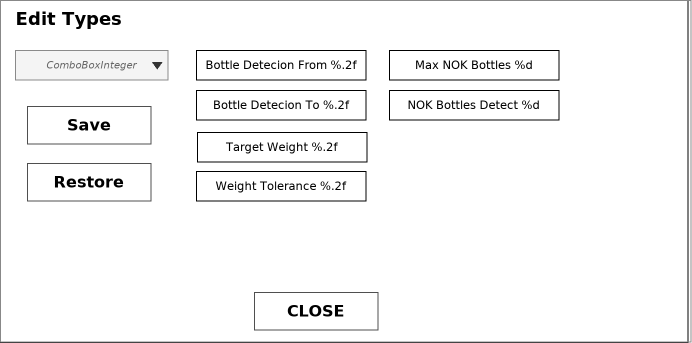
VISUALIZATION vTableEditTypes  // 692x343
VAR_IN_OUT
	fbTableControl: FB_TableControl;
END_VAR
    Rectangle (0,0 688x343)
    Label (-4,2 145x34), "Edit Types"
    Rectangle (254,292 124x38), "CLOSE"
        OnMouseDown: execute { fbTableControl.stHMI.iDialogNumber:=0; }
    ComboBoxInteger (15,50 153x30), variable: fbTableControl.stHMI.nEditedType, text list: 'tlBottleTypes'
    Rectangle (27,106 124x38), "Save"
        OnMouseDown: execute { fbTableControl.stHMI.bSave:=TRUE; }
    Rectangle (196,50 170x30), "Bottle Detecion From %.2f", text variable: fbTableControl.stHMI.stEditedType.stLoadingBottleParams.rLoadingDetectionFrom
        OnMouseClick: write the text variable via Default, min 0, max 32767, title 'Detection From', format %.2f
    Rectangle (196,90 170x30), "Bottle Detecion To %.2f", text variable: fbTableControl.stHMI.stEditedType.stLoadingBottleParams.rLoadingDetectionTo
        OnMouseClick: write the text variable via Default, min 0, max 32767, title 'Detection To', format %.2f
    Rectangle (27,163 124x38), "Restore"
        OnMouseDown: execute { fbTableControl.stHMI.bRestore:=TRUE; }
    Rectangle (197,132 170x30), "Target Weight %.2f", text variable: fbTableControl.stHMI.stEditedType.stWeighingBottleParams.rTargetWeight
        OnMouseClick: write the text variable via Default, min 0, max 2000, title 'Target Weight', format %.2f
    Rectangle (196,171 170x30), "Weight Tolerance %.2f", text variable: fbTableControl.stHMI.stEditedType.stWeighingBottleParams.rWeightTolerance
        OnMouseClick: write the text variable via Default, min 0, max 50, title 'Weight Tolerance', format %.2f
    Rectangle (389,50 170x30), "Max NOK Bottles %d", text variable: fbTableControl.stHMI.stEditedType.stWeighingBottleParams.iMaxNOK_Bottles
        OnMouseClick: write the text variable via Default, min 0, max 50, title 'Weight Tolerance', format %.2f
    Rectangle (389,90 170x30), "NOK Bottles Detect %d", text variable: fbTableControl.stHMI.stEditedType.stWeighingBottleParams.iNOK_BottlesSensorDetect
        OnMouseClick: write the text variable via Default, min 0, max 50, title 'Weight Tolerance', format %.2f
END_VISUALIZATION

(* stored: Version 1.1.0.1, ProductVersion 3.1.4024.15
   Visu vTableEditTypes: Id {76d1b110-9bc8-4034-b3ca-7f74ef13cc06} *)
